{attribute addProperty BoxType "IODEVICETYPE_ETHERCATPROT"}
{attribute addProperty Id "Beckhoff_EL1xxxBeckhoff_EL1xxx_A02C084E586527331.5Beckhoff_EL2xxxBeckhoff_EL2xxx_6D51086F228032850.375Beckhoff_EL3xxxBeckhoff_EL3xxx_68884AC1117621470.25Beckhoff_EL3xxx_0030Beckhoff_EL3xxx_0030_2D07FB6C1489186.125Beckhoff_EL4xxxBeckhoff_EL4xxx_B43A2050182952286.875Beckhoff_EL5xxxBeckhoff_EL5xxx_C80BAEFE179002237.5Beckhoff_EL6xxxBeckhoff_EL6xxx_F14D3E2E200052500.625Beckhoff_EL7xxxBeckhoff_EL7xxx_9130E37B122461530.75Beckhoff_EL9xxxBeckhoff_EL9xxx_842928EF6550818.75Beckhoff_EL15xxBeckhoff_EL15xx_DB59F57A3542442.75Beckhoff_EL19xxBeckhoff_EL19xx_39A0946F21827.25Beckhoff_EL25xxBeckhoff_EL25xx_19393863164322054Beckhoff_EL29xxBeckhoff_EL29xx_4C00A64E46458Beckhoff_EL30xxBeckhoff_EL30xx_21D80093342974287.125Beckhoff_EL31xxBeckhoff_EL31xx_0F318B7E188082351Beckhoff_EL32xxBeckhoff_EL32xx_64999344163342041.75Beckhoff_EL33xxBeckhoff_EL33xx_B84F5D38182282278.5Beckhoff_EL34xxBeckhoff_EL34xx_4C2EC3D09103811379.75Beckhoff_EL37xxBeckhoff_EL37xx_735867E2155961949.5Beckhoff_EL47xxBeckhoff_EL47xx_965E51942310288.75Beckhoff_EL66xxBeckhoff_EL66xx_C1E1F3707796974.5Beckhoff_EL67xxBeckhoff_EL67xx_2DE66D457644955.5Beckhoff_EL68xxBeckhoff_EL68xx_2DEB682D284623557.75Beckhoff_EL69xxBeckhoff_EL69xx_A41E28271430178.75Beckhoff_EL72xxBeckhoff_EL72xx_B1894506256363204.5Beckhoff_EL73xxBeckhoff_EL73xx_9CF0DC045462682.75Beckhoff_EL99xxBeckhoff_EL99xx_E89A1FE1526.5SyncUnitsSyncUnits_16C0B0F3134551681.875InputsInputs_C75D3FEC1280160OutputsOutputs_47D1E803848106InfoDataInfoData_E9F65A829612"}
{attribute addProperty CRC "3575571183"}
{attribute addProperty SizeInBites "479130"}
{attribute addProperty SizeInBytes "59891.25"}
TYPE EtherCAT_Master_ELxxxx_D51EE2EF :
STRUCT
	{attribute addProperty Name "Beckhoff_EL1xxx"}
	Beckhoff_EL1xxx : Beckhoff_EL1xxx_A02C084E;
	{attribute addProperty Name "Beckhoff_EL2xxx"}
	Beckhoff_EL2xxx : Beckhoff_EL2xxx_6D51086F;
	{attribute addProperty Name "Beckhoff_EL3xxx"}
	Beckhoff_EL3xxx : Beckhoff_EL3xxx_68884AC1;
	{attribute addProperty Name "Beckhoff_EL3xxx_0030"}
	Beckhoff_EL3xxx_0030 : Beckhoff_EL3xxx_0030_2D07FB6C;
	{attribute addProperty Name "Beckhoff_EL4xxx"}
	Beckhoff_EL4xxx : Beckhoff_EL4xxx_B43A2050;
	{attribute addProperty Name "Beckhoff_EL5xxx"}
	Beckhoff_EL5xxx : Beckhoff_EL5xxx_C80BAEFE;
	{attribute addProperty Name "Beckhoff_EL6xxx"}
	Beckhoff_EL6xxx : Beckhoff_EL6xxx_F14D3E2E;
	{attribute addProperty Name "Beckhoff_EL7xxx"}
	Beckhoff_EL7xxx : Beckhoff_EL7xxx_9130E37B;
	{attribute addProperty Name "Beckhoff_EL9xxx"}
	Beckhoff_EL9xxx : Beckhoff_EL9xxx_842928EF;
	{attribute addProperty Name "Beckhoff_EL15xx"}
	Beckhoff_EL15xx : Beckhoff_EL15xx_DB59F57A;
	{attribute addProperty Name "Beckhoff_EL19xx"}
	Beckhoff_EL19xx : Beckhoff_EL19xx_39A0946F;
	{attribute addProperty Name "Beckhoff_EL25xx"}
	Beckhoff_EL25xx : Beckhoff_EL25xx_19393863;
	{attribute addProperty Name "Beckhoff_EL29xx"}
	Beckhoff_EL29xx : Beckhoff_EL29xx_4C00A64E;
	{attribute addProperty Name "Beckhoff_EL30xx"}
	Beckhoff_EL30xx : Beckhoff_EL30xx_21D80093;
	{attribute addProperty Name "Beckhoff_EL31xx"}
	Beckhoff_EL31xx : Beckhoff_EL31xx_0F318B7E;
	{attribute addProperty Name "Beckhoff_EL32xx"}
	Beckhoff_EL32xx : Beckhoff_EL32xx_64999344;
	{attribute addProperty Name "Beckhoff_EL33xx"}
	Beckhoff_EL33xx : Beckhoff_EL33xx_B84F5D38;
	{attribute addProperty Name "Beckhoff_EL34xx"}
	Beckhoff_EL34xx : Beckhoff_EL34xx_4C2EC3D0;
	{attribute addProperty Name "Beckhoff_EL37xx"}
	Beckhoff_EL37xx : Beckhoff_EL37xx_735867E2;
	{attribute addProperty Name "Beckhoff_EL47xx"}
	Beckhoff_EL47xx : Beckhoff_EL47xx_965E5194;
	{attribute addProperty Name "Beckhoff_EL66xx"}
	Beckhoff_EL66xx : Beckhoff_EL66xx_C1E1F370;
	{attribute addProperty Name "Beckhoff_EL67xx"}
	Beckhoff_EL67xx : Beckhoff_EL67xx_2DE66D45;
	{attribute addProperty Name "Beckhoff_EL68xx"}
	Beckhoff_EL68xx : Beckhoff_EL68xx_2DEB682D;
	{attribute addProperty Name "Beckhoff_EL69xx"}
	Beckhoff_EL69xx : Beckhoff_EL69xx_A41E2827;
	{attribute addProperty Name "Beckhoff_EL72xx"}
	Beckhoff_EL72xx : Beckhoff_EL72xx_B1894506;
	{attribute addProperty Name "Beckhoff_EL73xx"}
	Beckhoff_EL73xx : Beckhoff_EL73xx_9CF0DC04;
	{attribute addProperty Name "Beckhoff_EL99xx"}
	Beckhoff_EL99xx : Beckhoff_EL99xx_E89A1FE1;
	{attribute addProperty Name "SyncUnits"}
	SyncUnits : SyncUnits_16C0B0F3;
	{attribute addProperty Name "Inputs"}
	Inputs : Inputs_C75D3FEC;
	{attribute addProperty Name "Outputs"}
	Outputs : Outputs_47D1E803;
	{attribute addProperty Name "InfoData"}
	InfoData : InfoData_E9F65A82;
END_STRUCT
END_TYPE

(* stored: Version 1.2.0.0, ProductVersion 3.1.4024.9
   DUT EtherCAT_Master_ELxxxx_D51EE2EF: Id {17bff535-3687-43c5-8c87-ae6aaee29005} *)
